{attribute 'qualified_only'}
{attribute 'strict'}
TYPE E_BoxPlaceDirection :
(
	UNDEFINED		:=  0,
	PLACE1_LEFT		:=	1,
	PLACE2_RIGHT	:=	2,
	
	LastPlace
);
END_TYPE

(* stored: Version 1.1.0.1, ProductVersion 3.1.4024.9
   DUT E_BoxPlaceDirection: Id {a41ea49e-68df-412f-aba6-c01a10f18526} *)
